PROGRAM PRG_FB_AnalogInput_Test
VAR
	bFirsCycle		: BOOL := TRUE;		(* First cycle flag *)
	
	rValue			: REAL;				(* Value from object property *)
	rValueForce		: REAL;				(* Value send to force method *)
	bSetForceValue 	: BOOL;				(* Enable forcing  *)
	
	rValueMin 		: REAL := 0.0;		(*  *)
	rValueMax		: REAL := 10.0;		(*  *)
	rChannelMin		: REAL := 0.0;		(*  *)
	rChannelMax		: REAL := 32767.0;	(*  *)
	
	fbAnalogInput 	: FB_AnalogInput;	(* Analog input object *)
END_VAR

(* Set properties *)
IF bFirsCycle THEN
	bFirsCycle := FALSE;
	fbAnalogInput.MR_FirstCycle( 	sName 			:= 'My test analog input',
									rValueScaledMin := rValueMin,
									rValueScaledMax := rValueMax,
									rChannelMin 	:= rChannelMin,
									rChannelMax 	:= rChannelMax);
END_IF

(* Enable to force channel value *)
IF bSetForceValue THEN
	fbAnalogInput.EnableForce := TRUE;
	fbAnalogInput.MR_SetForceValue(rValueForce);
ELSE
	fbAnalogInput.EnableForce := FALSE;
END_IF

(* Scaned value direct from FB *)
rValue := fbAnalogInput.Value;

fbAnalogInput.ChannelMin	:= rChannelMin;
fbAnalogInput.ChannelMax 	:= rChannelMax;
fbAnalogInput.ValueMin 		:= rValueMin;
fbAnalogInput.ValueMax 		:= rValueMax;
fbAnalogInput();

END_PROGRAM

(* stored: Version 1.1.0.1, ProductVersion 3.1.4024.9
   POU PRG_FB_AnalogInput_Test: Id {cc723b56-65f9-4441-ae21-caa7ac691231}, SpecialFunc None *)
